(*
SPDX-FileCopyrightText: © 2026 Oleksandr Tiutyk <trofimich@gmail.com>
SPDX-License-Identifier: MIT
License: https://opensource.org/license/mit
*)

(*!
<summary>Runs the OpenFramework test tree and the independent runner contract suite.</summary>
<description>Instances must not be copied because their test fixtures contain non-copyable state.</description>
*)

{attribute 'no_assign'}
{attribute 'no_explicit_call' := 'do not call this function block directly'}
FUNCTION_BLOCK TestAutomationController EXTENDS TOF_Automation.AutomationController<0>
VAR_STAT
	//! <summary>Class name shared by all instances of this function block.</summary>
	{attribute 'hide'} 
	_ClassName : STRING := __POUNAME();
END_VAR
VAR
	//! <summary>Checks the framework with a separate driver and direct ADS results.</summary>
	_TestRunnerTest : TestRunnerContractTest;

	//! <summary>Owns the I/O symbols and the fixture borrowed by the test runner.</summary>
	_IOModelsTest : IOModelsTestFixture;
	
	//! <summary>Runs the general OpenFramework.Testing regression suites.</summary>
	_JsonConfigurationRunner : JsonConfigurationTestRunner(ioModelsFixture := _IOModelsTest);
END_VAR

PROPERTY Children : REFERENCE TO ARRAY [0.._ChildCount - 1] OF TOF_Automation.IChildAutomationComponent
GET
Children REF= 0;
END_GET
END_PROPERTY

{attribute 'monitoring' := 'call'}
PROPERTY ClassName : REFERENCE TO STRING
GET
ClassName REF= _ClassName;
END_GET
END_PROPERTY

{attribute 'monitoring' := 'call'}
PROPERTY NamespaceName : REFERENCE TO STRING
GET
NamespaceName REF= CurrentNamespace.Name;
END_GET
END_PROPERTY

(*!
<summary>Advances filesystem test-root preparation, the independent contract suite, and the general test tree.</summary>
<description>
One controller task owns FileTestRoot. Suites observe its readiness instead of issuing competing root-create
requests. The independent suite has its own assertions and result reporting. AutomationRunner cleans task
memory after both test paths. Keep calling the controller so root and scenario cleanup can finish.
</description>
*)
METHOD PROTECTED OnBeforeChildrenWorking
VAR
	exceptionCode : __SYSTEM.ExceptionCode;
	exception : TOF_Core.IException;
	lastExMessage : TOF_Core.ERROR_MESSAGE;
	logMessage : STRING(255);
END_VAR
FileTestRoot.Execute();
_TestRunnerTest.Execute();

__TRY
	_JsonConfigurationRunner.Execute(cleanupTaskMemory := FALSE);
__CATCH(exceptionCode)
	exception := TOF_Core.ExceptionManager.GetLastException(
		exceptionCode := exceptionCode,
		catchPointNamespaceName := NamespaceName,
		catchPointPOUName := __POUNAME(),
		catchPointPosition := __POSITION()
	);
	lastExMessage := exception.GetMessage(
		showSource := TRUE,
		timestampDisplayMode := TOF_Core.TIMESTAMP_DISPLAY_MODE.LOCAL
	);
	logMessage := TO_STRING(lastExMessage);

	Tc2_System.ADSLOGSTR(
		msgCtrlMask := Tc2_System.Global_Variables.ADSLOG_MSGTYPE_ERROR,
		msgFmtStr := 'CRITICAL: _JsonConfigurationRunner threw: %s',
		strArg := logMessage
	);

	TOF_Core.ExceptionManager.ReThrowLastException(
		exceptionCode := exceptionCode,
		catchPointNamespaceName := NamespaceName,
		catchPointPOUName := __POUNAME(),
		catchPointPosition := __POSITION()
	);
__ENDTRY
END_METHOD

{attribute 'monitoring' := 'call'}
PROPERTY SelfSize : ULINT
GET
SelfSize := XSIZEOF(THIS^);
END_GET
END_PROPERTY

{attribute 'monitoring' := 'call'}
PROPERTY StartRequest : BOOL
GET
StartRequest := TRUE;
END_GET
END_PROPERTY

END_FUNCTION_BLOCK

(* stored: Version 1.1.0.1, ProductVersion 3.1.4026.21
   POU TestAutomationController: Id {66626e70-d017-4266-8769-7cd39f80d94d}, SpecialFunc None
   Property Children: Id {808e2bb2-4cf4-4bed-af77-c4b90dfaf272}
   Get Get: Id {68e5d592-b357-4d3f-a459-568d988331ee}
   Property ClassName: Id {9a23e807-4502-4ff5-a340-bb5707bed577}
   Get Get: Id {48e70ac4-e138-48c7-8d5b-78bb20caab4a}
   Property NamespaceName: Id {9ca5477b-09fe-4c45-990a-565a2307423e}
   Get Get: Id {c5c86d10-aae1-44b0-b97e-fba9982acf76}
   Method OnBeforeChildrenWorking: Id {f0394797-3eeb-44c9-847b-75920f0bbead}
   Property SelfSize: Id {f40e5ad6-7a53-4a63-913b-db682a7c26c5}
   Get Get: Id {b6cba390-e08d-46b6-8503-4a7f2b18b1a3}
   Property StartRequest: Id {51469ead-ef1f-4035-91bd-fc88dd6dc76f}
   Get Get: Id {85844015-c398-4fea-800c-924fcc442941} *)
